TYPE ST_UserControlGrid_FromHmi :
STRUCT
	stButtonSave	: ST_HMI_BUTTON_IN;
END_STRUCT
END_TYPE

(* stored: Version 1.1.0.1, ProductVersion 3.1.4024.11
   DUT ST_UserControlGrid_FromHmi: Id {3f19c66e-538e-40b6-bb26-7a95ee61d41d} *)
